{attribute 'linkalways'} 
{attribute 'no_explicit_call' := 'This FB is a CLASS and must be accessed using methods or properties'}
{attribute 'enable_dynamic_creation'}
FUNCTION_BLOCK _INT EXTENDS NumericDatatypeBase
VAR
	localData : INT;
	activeData : REFERENCE TO INT REF= localData;
END_VAR

PROPERTY PUBLIC Address : PVOID
GET
Address := ADR(activeData);
END_GET
END_PROPERTY

METHOD PUBLIC ClearReference
VAR_INPUT
END_VAR
activeData REF= localData;
END_METHOD

METHOD PUBLIC Clone : I_Datatype
VAR
    pClone : POINTER TO _INT;
END_VAR
pClone := __NEW(_INT(InitialValue := Value));
Clone := pClone^;
END_METHOD

METHOD FB_init : BOOL
VAR_INPUT
	bInitRetains : BOOL; // if TRUE, the retain variables are initialized (warm start / cold start)
	bInCopyCode : BOOL;  // if TRUE, the instance afterwards gets moved into the copy code (online change)
	InitialValue : INT;
END_VAR
localData := InitialValue;
END_METHOD

PROPERTY PUBLIC IsFloat : BOOL
GET
IsFloat := FALSE;
END_GET
END_PROPERTY

PROPERTY PUBLIC IsSigned : BOOL
GET
IsSigned := TRUE;
END_GET
END_PROPERTY

METHOD PUBLIC MakeReferenceTo
VAR_INPUT
	ReferenceTarget : REFERENCE TO INT;
END_VAR
activeData REF= ReferenceTarget;
END_METHOD

PROPERTY PUBLIC MaxValue : INT
GET
MaxValue := DatatypeLimits.INT_MAX_VALUE;
END_GET
END_PROPERTY

PROPERTY PUBLIC MinValue : INT
GET
MinValue := DatatypeLimits.INT_MIN_VALUE;
END_GET
END_PROPERTY

METHOD PROTECTED SerializeMaxValue
VAR_INPUT
	Serializer : I_Serializer;
END_VAR
Serializer.AddInt(MaxValue);
END_METHOD

METHOD PROTECTED SerializeMinValue
VAR_INPUT
	Serializer : I_Serializer;
END_VAR
Serializer.AddInt(MinValue);
END_METHOD

METHOD PUBLIC SerializeWith
VAR_INPUT
	Serializer : I_Serializer;
END_VAR
Serializer.AddInt(activeData);
END_METHOD

PROPERTY PUBLIC Size : UDINT
GET
Size := SIZEOF(activeData);
END_GET
END_PROPERTY

METHOD TryDeserializeFrom : BOOL
VAR_INPUT
	Deserializer : I_Deserializer;
	Feedback : I_DeserializerFeedback;
END_VAR
TryDeserializeFrom := Deserializer.TryGetInt(activeData, Feedback);
END_METHOD

METHOD TryMakeReferenceTo : BOOL
VAR_INPUT
	Target : I_Datatype;
END_VAR
VAR
	pTargetData : POINTER TO INT;
END_VAR
IF NOT (Target.TypeName = TypeName) THEN
	RETURN;
END_IF

pTargetData := Target.Address;
activeData REF= pTargetData^;
TryMakeReferenceTo := TRUE;
END_METHOD

PROPERTY PUBLIC TypeName : T_MAXSTRING
GET
TypeName := 'INT';
END_GET
END_PROPERTY

PROPERTY PUBLIC Value : REFERENCE TO INT
GET
Value REF= activeData;
END_GET
END_PROPERTY

END_FUNCTION_BLOCK

(* stored: Version 1.1.0.1, ProductVersion 3.1.4024.12
   POU _INT: Id {41ebb93b-a842-465a-bbf3-cd64336e2c9d}, SpecialFunc None
   Folder Constructor: Id {33715b41-23bb-45de-a8df-702b4ae01469}
   Folder Protected: Id {19fcd262-ac7a-47eb-8b95-8ed109346db4}
   Property Address: Id {3f13b4b2-c59d-475f-be30-646f489b8d11}
   Get Get: Id {abfd6187-bd6d-4bd7-af15-918241af3f39}
   Method ClearReference: Id {715b0508-849f-4314-8f18-0e7d903a3b05}
   Method Clone: Id {c754c0f7-22d0-433a-aed2-a1d47ec47913}
   Method FB_init: Id {cdf4dda5-fa59-4f4c-a218-d23983f318cd}
   Property IsFloat: Id {cf49872e-156d-45c8-ad81-0a5594298cee}
   Get Get: Id {482ddbc7-1562-46ce-babe-d0625f464472}
   Property IsSigned: Id {80d3994b-4b84-416b-93b1-665f7204395e}
   Get Get: Id {f61b45fc-3075-4363-af81-1ffbb7afc885}
   Method MakeReferenceTo: Id {ac18a1da-f36c-4964-989c-90e2a586a86a}
   Property MaxValue: Id {e1eae55b-04e2-425b-8924-32c66298ae0b}
   Get Get: Id {eda88a0d-6f6a-4dcd-b83d-1976ba9f3edb}
   Property MinValue: Id {cf50978f-7672-4e8f-8d98-bcb30a305e25}
   Get Get: Id {5e8c3705-2503-445e-b4c5-81053687a72e}
   Method SerializeMaxValue: Id {52a3144f-84b0-414e-a087-0a7b1dfde97f}
   Method SerializeMinValue: Id {38e40e28-6ea9-46dc-86c5-bef8cff7eda4}
   Method SerializeWith: Id {09b3f5be-fb97-469c-a8fe-5605e9743cbc}
   Property Size: Id {6baf373f-eb31-4715-b539-54888fd8273a}
   Get Get: Id {2f0c7348-7a2c-484a-bd4d-e69f750f518e}
   Method TryDeserializeFrom: Id {e3f8c69d-2382-4b8a-b50d-566bcafa87d7}
   Method TryMakeReferenceTo: Id {e81878de-45cb-4854-b63a-a0c0e77f920a}
   Property TypeName: Id {b6db8aed-06e2-402d-ba79-825fbfdd297c}
   Get Get: Id {8be2b323-a4d2-4c78-9c38-8d095b769687}
   Property Value: Id {2882c603-557d-4cba-a6f8-b35e21afd466}
   Get Get: Id {35fd66eb-14df-42e3-9529-f03f550f961e} *)
